// TIA Portal V16 export
// export: Created 2024-09-05T17:39:09.8002543Z, ExportSetting WithDefaults, DisplayName Totally Integrated Automation Portal, DisplayVersion V16 Update 6, DisplayName TIA Portal Version Control Interface, DisplayVersion V16 Update 2, DisplayName TIA Portal Openness, DisplayVersion V16 Update 6, DisplayName STEP 7 Professional, DisplayVersion V16 Update 6, DisplayName STEP 7 Safety, DisplayVersion V16, DisplayName WinCC Advanced, DisplayVersion V16 Update 6
FUNCTION_BLOCK "FittingCycle"   // FB35, LAD
{ S7_Optimized_Access := 'TRUE' }
VERSION : 0.1
// stored: AutoNumber true, IsIECCheckEnabled false, IsRetainMemResEnabled false, MemoryReserve 100, SetENOAutomatically false, UDAEnableTagReadback false
   VAR_INPUT
      parameters : "UDT_FittingParameters";
      basicPosition : Bool;
      MaxPosition : Real;
      endStopCylinderActive : Bool;
      shiftSupportToWork : Bool;
      rivetSensor : Bool;
      rivetStatusOtherCylinder : SInt;
   END_VAR
   VAR_IN_OUT
      HydraulicCylinder : "UDT_HydraulicCylinderData";
      dataFitting : "UDT_FittingStatus";
      dataDigiforce : "UDT_Digiforce";
      stopperForWedgeCylinder : "UDT_Cylinder";
      supportCylinder : "UDT_Cylinder";
      wedgeCylinder : "UDT_Cylinder";
      MeasuredData : "UDT_Results_Cupforming";
   END_VAR
   VAR
      cnt : Int;
      R_TRIG_Instance { S7_SetPoint := 'True'} : R_TRIG;
      H2Reached { S7_SetPoint := 'True'} : Bool;
      IEC_Timer_timeout { S7_SetPoint := 'True'} : TON_TIME;
      DigiforceStarted { S7_SetPoint := 'True'} : Bool;
      R_TRIG_Instance_1 { S7_SetPoint := 'True'} : R_TRIG;
      ton_WayWithTimeoutReached { S7_SetPoint := 'True'} : TON_TIME;
   END_VAR
   VAR_TEMP   // added for the SCL form of the ladder/FBD networks
      _w1 : Bool;
      _w2 : Bool;
   END_VAR
BEGIN

REGION Network 1: Check min max values
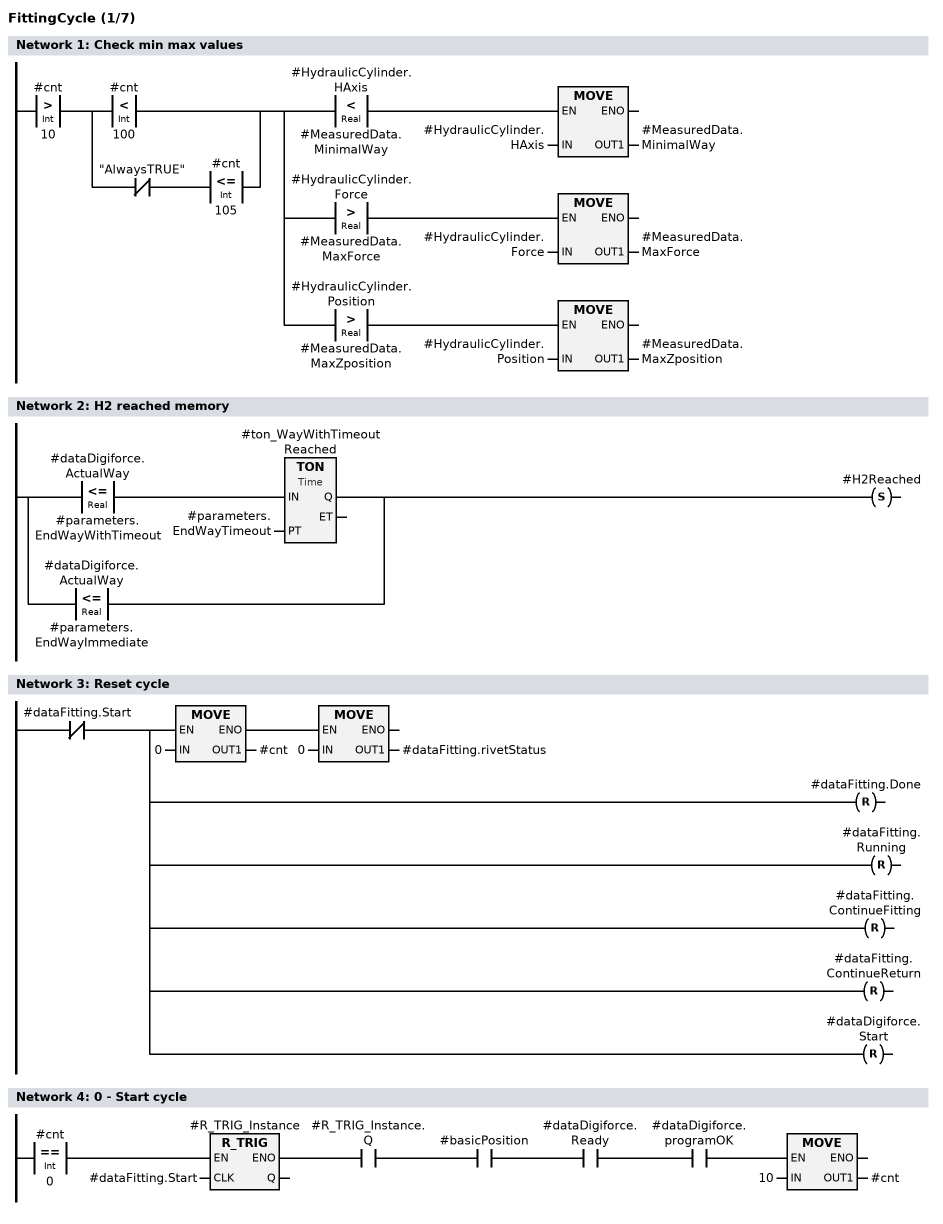
   RUNG wire#powerrail
      { S7_Templates := "SrcType := Int" } GT_Contact(in1 := #cnt, in2 := 10)
      wire#w1
      { S7_Templates := "SrcType := Int" } LT_Contact(in1 := #cnt, in2 := 100)
      wire#w2
      { S7_Templates := "SrcType := Real" } LT_Contact(in1 := #HydraulicCylinder.HAxis, in2 := #MeasuredData.MinimalWay)
      Move(in := #HydraulicCylinder.HAxis, out1 => #MeasuredData.MinimalWay)
   END_RUNG
   RUNG wire#w1
      I_Contact( "AlwaysTRUE" )
      { S7_Templates := "SrcType := Int" } LE_Contact(in1 := #cnt, in2 := 105)
   END_RUNG wire#w2
   RUNG wire#w2
      { S7_Templates := "SrcType := Real" } GT_Contact(in1 := #HydraulicCylinder.Force, in2 := #MeasuredData.MaxForce)
      Move(in := #HydraulicCylinder.Force, out1 => #MeasuredData.MaxForce)
   END_RUNG
   RUNG wire#w2
      { S7_Templates := "SrcType := Real" } GT_Contact(in1 := #HydraulicCylinder.Position, in2 := #MeasuredData.MaxZposition)
      Move(in := #HydraulicCylinder.Position, out1 => #MeasuredData.MaxZposition)
   END_RUNG
   // the same network as SCL:
   #_w1 := (#cnt > 10) AND ((#cnt < 100) OR (NOT "AlwaysTRUE" AND (#cnt <= 105)));
   IF #_w1 AND (#HydraulicCylinder.HAxis < #MeasuredData.MinimalWay) THEN
       #MeasuredData.MinimalWay := #HydraulicCylinder.HAxis;
   END_IF;
   IF #_w1 AND (#HydraulicCylinder.Force > #MeasuredData.MaxForce) THEN
       #MeasuredData.MaxForce := #HydraulicCylinder.Force;
   END_IF;
   IF #_w1 AND (#HydraulicCylinder.Position > #MeasuredData.MaxZposition) THEN
       #MeasuredData.MaxZposition := #HydraulicCylinder.Position;
   END_IF;
END_REGION

REGION Network 2: H2 reached memory
   RUNG wire#powerrail
      { S7_Templates := "SrcType := Real" } LE_Contact(in1 := #dataDigiforce.ActualWay, in2 := #parameters.EndWayWithTimeout)
      { S7_Templates := "time_type := Time" } #ton_WayWithTimeoutReached.TON(pt := #parameters.EndWayTimeout, et =>)
      wire#w1
      S_Coil( #H2Reached )
   END_RUNG
   RUNG wire#powerrail
      { S7_Templates := "SrcType := Real" } LE_Contact(in1 := #dataDigiforce.ActualWay, in2 := #parameters.EndWayImmediate)
   END_RUNG wire#w1
   // the same network as SCL:
   #ton_WayWithTimeoutReached(IN := #dataDigiforce.ActualWay <= #parameters.EndWayWithTimeout,   // TON
                           PT := #parameters.EndWayTimeout);
   IF #ton_WayWithTimeoutReached.Q OR (#dataDigiforce.ActualWay <= #parameters.EndWayImmediate) THEN
       #H2Reached := TRUE;
   END_IF;
END_REGION

REGION Network 3: Reset cycle
   RUNG wire#powerrail
      I_Contact( #dataFitting.Start )
      wire#w1
      Move(in := 0, out1 => #cnt)
      Move(in := 0, out1 => #dataFitting.rivetStatus)
   END_RUNG
   RUNG wire#w1
      R_Coil( #dataFitting.Done )
   END_RUNG
   RUNG wire#w1
      R_Coil( #dataFitting.Running )
   END_RUNG
   RUNG wire#w1
      R_Coil( #dataFitting.ContinueFitting )
   END_RUNG
   RUNG wire#w1
      R_Coil( #dataFitting.ContinueReturn )
   END_RUNG
   RUNG wire#w1
      R_Coil( #dataDigiforce.Start )
   END_RUNG
   // the same network as SCL:
   IF NOT #dataFitting.Start THEN
       #cnt := 0;
       #dataFitting.rivetStatus := 0;
       #dataFitting.Done := FALSE;
       #dataFitting.Running := FALSE;
       #dataFitting.ContinueFitting := FALSE;
       #dataFitting.ContinueReturn := FALSE;
       #dataDigiforce.Start := FALSE;
   END_IF;
END_REGION

REGION Network 4: 0 - Start cycle
   RUNG wire#powerrail
      { S7_Templates := "SrcType := Int" } EQ_Contact(in1 := #cnt, in2 := 0)
      #R_TRIG_Instance.R_TRIG(CLK := #dataFitting.Start, Q =>)
      Contact( #R_TRIG_Instance.Q )
      Contact( #basicPosition )
      Contact( #dataDigiforce.Ready )
      Contact( #dataDigiforce.programOK )
      Move(in := 10, out1 => #cnt)
   END_RUNG
   // the same network as SCL:
   #_w1 := #cnt = 0;
   #R_TRIG_Instance(EN := #_w1, CLK := #dataFitting.Start, ENO => #_w2);   // R_TRIG
   IF #_w2 AND #R_TRIG_Instance.Q AND #basicPosition AND #dataDigiforce.Ready AND #dataDigiforce.programOK THEN
       #cnt := 10;
   END_IF;
END_REGION

REGION Network 5: 10 - Start cycle
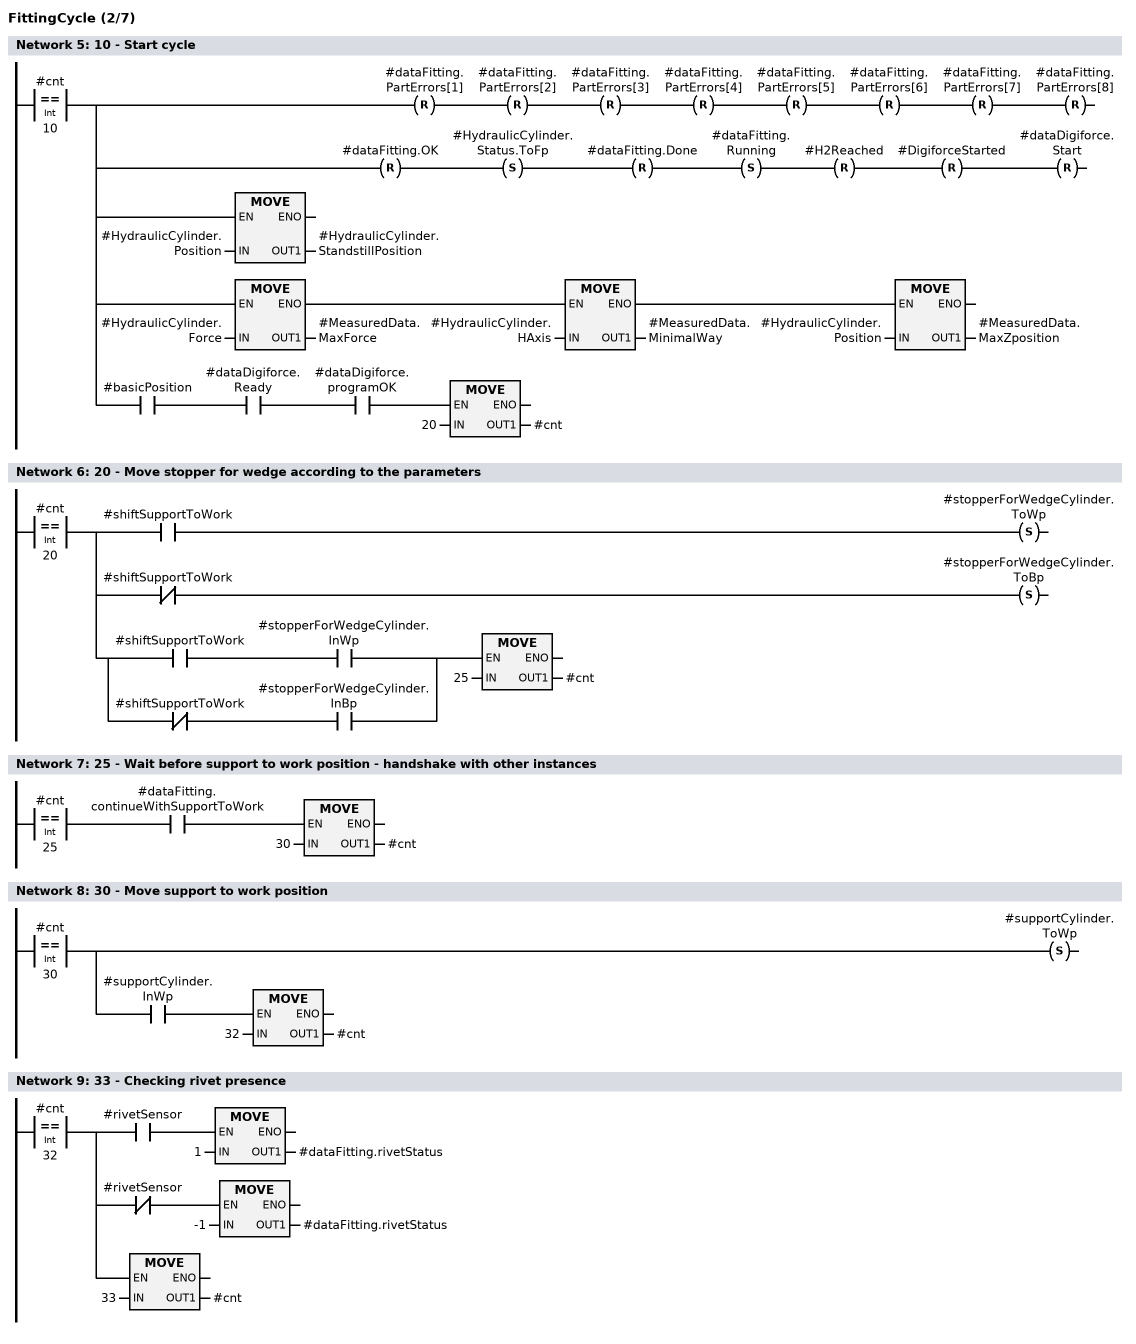
   RUNG wire#powerrail
      { S7_Templates := "SrcType := Int" } EQ_Contact(in1 := #cnt, in2 := 10)
      wire#w1
      R_Coil( #dataFitting.PartErrors[1] )
      R_Coil( #dataFitting.PartErrors[2] )
      R_Coil( #dataFitting.PartErrors[3] )
      R_Coil( #dataFitting.PartErrors[4] )
      R_Coil( #dataFitting.PartErrors[5] )
      R_Coil( #dataFitting.PartErrors[6] )
      R_Coil( #dataFitting.PartErrors[7] )
      R_Coil( #dataFitting.PartErrors[8] )
   END_RUNG
   RUNG wire#w1
      R_Coil( #dataFitting.OK )
      S_Coil( #HydraulicCylinder.Status.ToFp )
      R_Coil( #dataFitting.Done )
      S_Coil( #dataFitting.Running )
      R_Coil( #H2Reached )
      R_Coil( #DigiforceStarted )
      R_Coil( #dataDigiforce.Start )
   END_RUNG
   RUNG wire#w1
      Move(in := #HydraulicCylinder.Position, out1 => #HydraulicCylinder.StandstillPosition)
   END_RUNG
   RUNG wire#w1
      Move(in := #HydraulicCylinder.Force, out1 => #MeasuredData.MaxForce)
      Move(in := #HydraulicCylinder.HAxis, out1 => #MeasuredData.MinimalWay)
      Move(in := #HydraulicCylinder.Position, out1 => #MeasuredData.MaxZposition)
   END_RUNG
   RUNG wire#w1
      Contact( #basicPosition )
      Contact( #dataDigiforce.Ready )
      Contact( #dataDigiforce.programOK )
      Move(in := 20, out1 => #cnt)
   END_RUNG
   // the same network as SCL:
   #_w1 := #cnt = 10;
   IF #_w1 THEN
       #dataFitting.PartErrors[1] := FALSE;
       #dataFitting.PartErrors[2] := FALSE;
       #dataFitting.PartErrors[3] := FALSE;
       #dataFitting.PartErrors[4] := FALSE;
       #dataFitting.PartErrors[5] := FALSE;
       #dataFitting.PartErrors[6] := FALSE;
       #dataFitting.PartErrors[7] := FALSE;
       #dataFitting.PartErrors[8] := FALSE;
       #dataFitting.OK := FALSE;
       #HydraulicCylinder.Status.ToFp := TRUE;
       #dataFitting.Done := FALSE;
       #dataFitting.Running := TRUE;
       #H2Reached := FALSE;
       #DigiforceStarted := FALSE;
       #dataDigiforce.Start := FALSE;
       #HydraulicCylinder.StandstillPosition := #HydraulicCylinder.Position;
       #MeasuredData.MaxForce := #HydraulicCylinder.Force;
       #MeasuredData.MinimalWay := #HydraulicCylinder.HAxis;
       #MeasuredData.MaxZposition := #HydraulicCylinder.Position;
   END_IF;
   IF #_w1 AND #basicPosition AND #dataDigiforce.Ready AND #dataDigiforce.programOK THEN #cnt := 20; END_IF;
END_REGION

REGION Network 6: 20 - Move stopper for wedge according to the parameters
   RUNG wire#powerrail
      { S7_Templates := "SrcType := Int" } EQ_Contact(in1 := #cnt, in2 := 20)
      wire#w1
      Contact( #shiftSupportToWork )
      S_Coil( #stopperForWedgeCylinder.ToWp )
   END_RUNG
   RUNG wire#w1
      I_Contact( #shiftSupportToWork )
      S_Coil( #stopperForWedgeCylinder.ToBp )
   END_RUNG
   RUNG wire#w1
      Contact( #shiftSupportToWork )
      Contact( #stopperForWedgeCylinder.InWp )
      wire#w2
      Move(in := 25, out1 => #cnt)
   END_RUNG
   RUNG wire#w1
      I_Contact( #shiftSupportToWork )
      Contact( #stopperForWedgeCylinder.InBp )
   END_RUNG wire#w2
   // the same network as SCL:
   #_w1 := #cnt = 20;
   IF #_w1 AND #shiftSupportToWork THEN #stopperForWedgeCylinder.ToWp := TRUE; END_IF;
   IF #_w1 AND NOT #shiftSupportToWork THEN #stopperForWedgeCylinder.ToBp := TRUE; END_IF;
   IF #_w1 AND ((#shiftSupportToWork AND #stopperForWedgeCylinder.InWp) OR (NOT #shiftSupportToWork AND #stopperForWedgeCylinder.InBp)) THEN
       #cnt := 25;
   END_IF;
END_REGION

REGION Network 7: 25 - Wait before support to work position - handshake with other instances
   RUNG wire#powerrail
      { S7_Templates := "SrcType := Int" } EQ_Contact(in1 := #cnt, in2 := 25)
      Contact( #dataFitting.continueWithSupportToWork )
      Move(in := 30, out1 => #cnt)
   END_RUNG
   // the same network as SCL:
   IF (#cnt = 25) AND #dataFitting.continueWithSupportToWork THEN #cnt := 30; END_IF;
END_REGION

REGION Network 8: 30 - Move support to work position
   RUNG wire#powerrail
      { S7_Templates := "SrcType := Int" } EQ_Contact(in1 := #cnt, in2 := 30)
      wire#w1
      S_Coil( #supportCylinder.ToWp )
   END_RUNG
   RUNG wire#w1
      Contact( #supportCylinder.InWp )
      Move(in := 32, out1 => #cnt)
   END_RUNG
   // the same network as SCL:
   #_w1 := #cnt = 30;
   IF #_w1 THEN #supportCylinder.ToWp := TRUE; END_IF;
   IF #_w1 AND #supportCylinder.InWp THEN #cnt := 32; END_IF;
END_REGION

REGION Network 9: 33 - Checking rivet presence
   RUNG wire#powerrail
      { S7_Templates := "SrcType := Int" } EQ_Contact(in1 := #cnt, in2 := 32)
      wire#w1
      Contact( #rivetSensor )
      Move(in := 1, out1 => #dataFitting.rivetStatus)
   END_RUNG
   RUNG wire#w1
      I_Contact( #rivetSensor )
      Move(in := -1, out1 => #dataFitting.rivetStatus)
   END_RUNG
   RUNG wire#w1
      Move(in := 33, out1 => #cnt)
   END_RUNG
   // the same network as SCL:
   #_w1 := #cnt = 32;
   IF #_w1 AND #rivetSensor THEN #dataFitting.rivetStatus := 1; END_IF;
   IF #_w1 AND NOT #rivetSensor THEN #dataFitting.rivetStatus := -1; END_IF;
   IF #_w1 THEN #cnt := 33; END_IF;
END_REGION

REGION Network 10: 34 - Rivet presence result / handshake
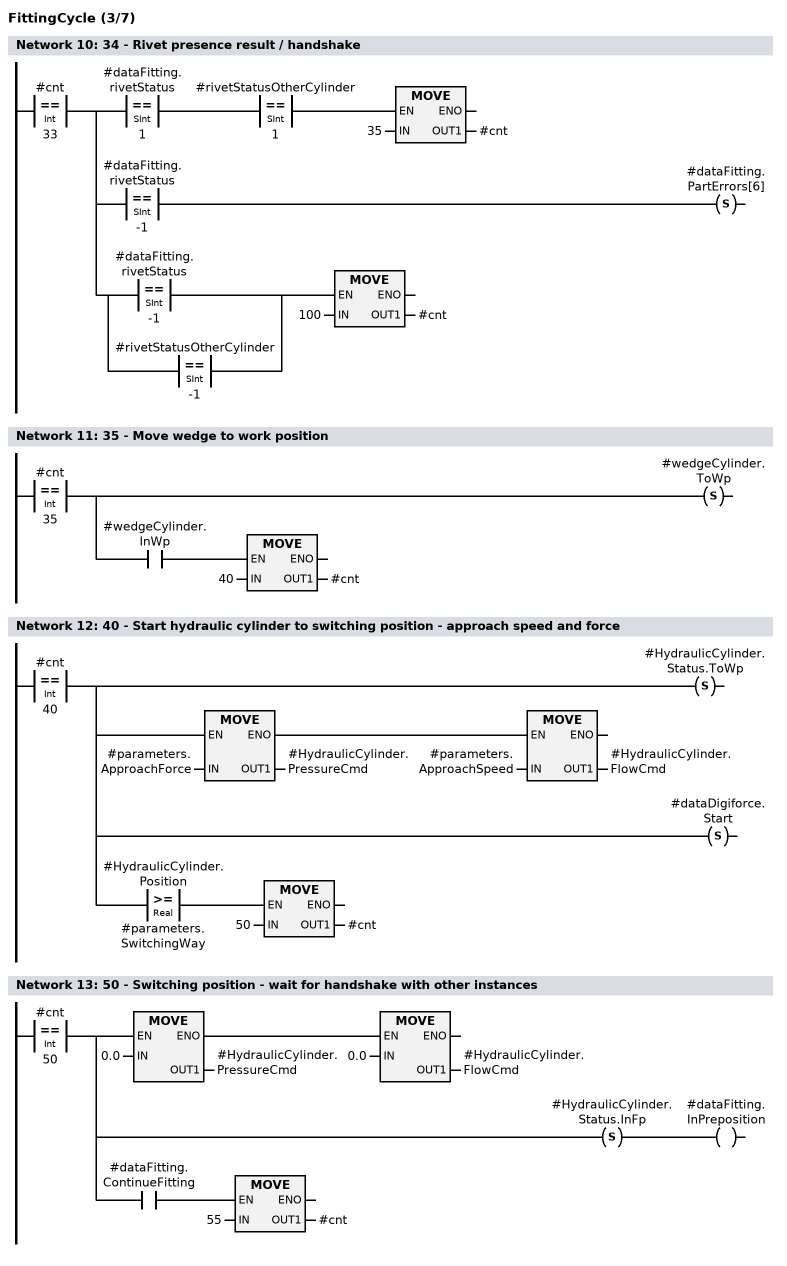
   RUNG wire#powerrail
      { S7_Templates := "SrcType := Int" } EQ_Contact(in1 := #cnt, in2 := 33)
      wire#w1
      { S7_Templates := "SrcType := SInt" } EQ_Contact(in1 := #dataFitting.rivetStatus, in2 := 1)
      { S7_Templates := "SrcType := SInt" } EQ_Contact(in1 := #rivetStatusOtherCylinder, in2 := 1)
      Move(in := 35, out1 => #cnt)
   END_RUNG
   RUNG wire#w1
      { S7_Templates := "SrcType := SInt" } EQ_Contact(in1 := #dataFitting.rivetStatus, in2 := -1)
      S_Coil( #dataFitting.PartErrors[6] )
   END_RUNG
   RUNG wire#w1
      { S7_Templates := "SrcType := SInt" } EQ_Contact(in1 := #dataFitting.rivetStatus, in2 := -1)
      wire#w2
      Move(in := 100, out1 => #cnt)
   END_RUNG
   RUNG wire#w1
      { S7_Templates := "SrcType := SInt" } EQ_Contact(in1 := #rivetStatusOtherCylinder, in2 := -1)
   END_RUNG wire#w2
   // the same network as SCL:
   #_w1 := #cnt = 33;
   IF #_w1 AND (#dataFitting.rivetStatus = 1) AND (#rivetStatusOtherCylinder = 1) THEN #cnt := 35; END_IF;
   IF #_w1 AND (#dataFitting.rivetStatus = (-1)) THEN #dataFitting.PartErrors[6] := TRUE; END_IF;
   IF #_w1 AND ((#dataFitting.rivetStatus = (-1)) OR (#rivetStatusOtherCylinder = (-1))) THEN
       #cnt := 100;
   END_IF;
END_REGION

REGION Network 11: 35 - Move wedge to work position
   RUNG wire#powerrail
      { S7_Templates := "SrcType := Int" } EQ_Contact(in1 := #cnt, in2 := 35)
      wire#w1
      S_Coil( #wedgeCylinder.ToWp )
   END_RUNG
   RUNG wire#w1
      Contact( #wedgeCylinder.InWp )
      Move(in := 40, out1 => #cnt)
   END_RUNG
   // the same network as SCL:
   #_w1 := #cnt = 35;
   IF #_w1 THEN #wedgeCylinder.ToWp := TRUE; END_IF;
   IF #_w1 AND #wedgeCylinder.InWp THEN #cnt := 40; END_IF;
END_REGION

REGION Network 12: 40 - Start hydraulic cylinder to switching position - approach speed and force
   RUNG wire#powerrail
      { S7_Templates := "SrcType := Int" } EQ_Contact(in1 := #cnt, in2 := 40)
      wire#w1
      S_Coil( #HydraulicCylinder.Status.ToWp )
   END_RUNG
   RUNG wire#w1
      Move(in := #parameters.ApproachForce, out1 => #HydraulicCylinder.PressureCmd)
      Move(in := #parameters.ApproachSpeed, out1 => #HydraulicCylinder.FlowCmd)
   END_RUNG
   RUNG wire#w1
      S_Coil( #dataDigiforce.Start )
   END_RUNG
   RUNG wire#w1
      { S7_Templates := "SrcType := Real" } GE_Contact(in1 := #HydraulicCylinder.Position, in2 := #parameters.SwitchingWay)
      Move(in := 50, out1 => #cnt)
   END_RUNG
   // the same network as SCL:
   #_w1 := #cnt = 40;
   IF #_w1 THEN
       #HydraulicCylinder.Status.ToWp := TRUE;
       #HydraulicCylinder.PressureCmd := #parameters.ApproachForce;
       #HydraulicCylinder.FlowCmd := #parameters.ApproachSpeed;
       #dataDigiforce.Start := TRUE;
   END_IF;
   IF #_w1 AND (#HydraulicCylinder.Position >= #parameters.SwitchingWay) THEN #cnt := 50; END_IF;
END_REGION

REGION Network 13: 50 - Switching position - wait for handshake with other instances
   RUNG wire#powerrail
      { S7_Templates := "SrcType := Int" } EQ_Contact(in1 := #cnt, in2 := 50)
      wire#w1
      Move(in := 0.0, out1 => #HydraulicCylinder.PressureCmd)
      Move(in := 0.0, out1 => #HydraulicCylinder.FlowCmd)
   END_RUNG
   RUNG wire#w1
      S_Coil( #HydraulicCylinder.Status.InFp )
      Coil( #dataFitting.InPreposition )
   END_RUNG
   RUNG wire#w1
      Contact( #dataFitting.ContinueFitting )
      Move(in := 55, out1 => #cnt)
   END_RUNG
   // the same network as SCL:
   #_w1 := #cnt = 50;
   IF #_w1 THEN
       #HydraulicCylinder.PressureCmd := 0.0;
       #HydraulicCylinder.FlowCmd := 0.0;
       #HydraulicCylinder.Status.InFp := TRUE;
   END_IF;
   #dataFitting.InPreposition := #_w1;
   IF #_w1 AND #dataFitting.ContinueFitting THEN #cnt := 55; END_IF;
END_REGION

REGION Network 14: 55 - Move sidemember to work position
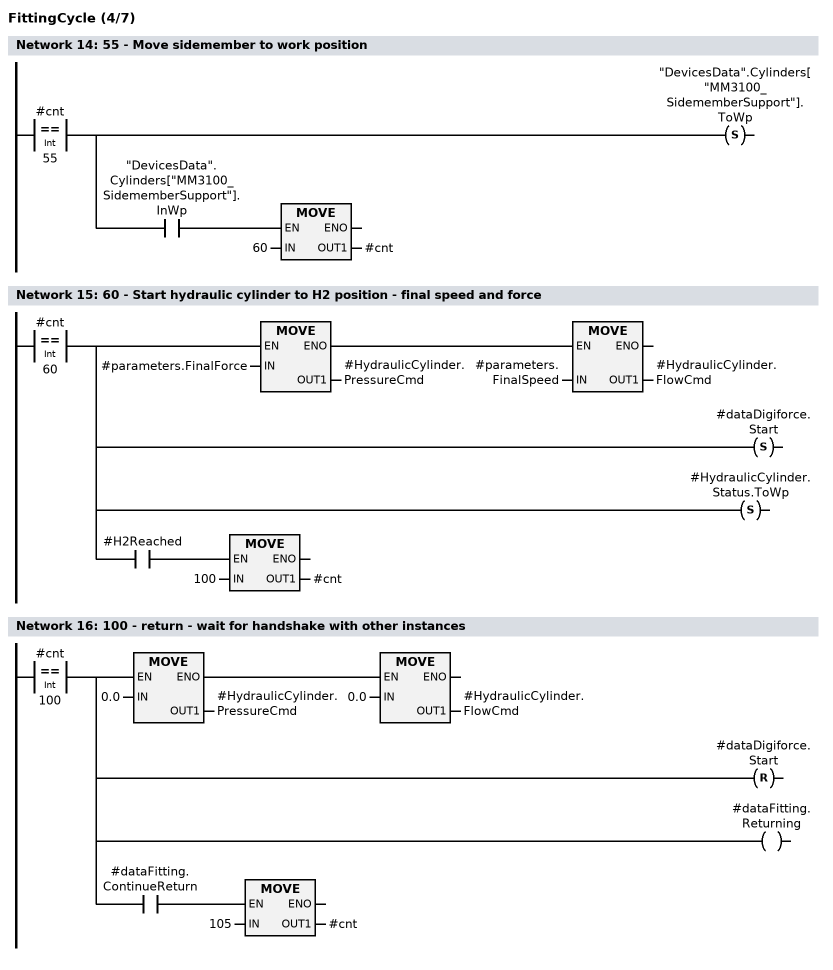
   RUNG wire#powerrail
      { S7_Templates := "SrcType := Int" } EQ_Contact(in1 := #cnt, in2 := 55)
      wire#w1
      S_Coil( "DevicesData".Cylinders["MM3100_SidememberSupport"].ToWp )
   END_RUNG
   RUNG wire#w1
      Contact( "DevicesData".Cylinders["MM3100_SidememberSupport"].InWp )
      Move(in := 60, out1 => #cnt)
   END_RUNG
   // the same network as SCL:
   #_w1 := #cnt = 55;
   IF #_w1 THEN "DevicesData".Cylinders["MM3100_SidememberSupport"].ToWp := TRUE; END_IF;
   IF #_w1 AND "DevicesData".Cylinders["MM3100_SidememberSupport"].InWp THEN #cnt := 60; END_IF;
END_REGION

REGION Network 15: 60 - Start hydraulic cylinder to H2 position - final speed and force
   RUNG wire#powerrail
      { S7_Templates := "SrcType := Int" } EQ_Contact(in1 := #cnt, in2 := 60)
      wire#w1
      Move(in := #parameters.FinalForce, out1 => #HydraulicCylinder.PressureCmd)
      Move(in := #parameters.FinalSpeed, out1 => #HydraulicCylinder.FlowCmd)
   END_RUNG
   RUNG wire#w1
      S_Coil( #dataDigiforce.Start )
   END_RUNG
   RUNG wire#w1
      S_Coil( #HydraulicCylinder.Status.ToWp )
   END_RUNG
   RUNG wire#w1
      Contact( #H2Reached )
      Move(in := 100, out1 => #cnt)
   END_RUNG
   // the same network as SCL:
   #_w1 := #cnt = 60;
   IF #_w1 THEN
       #HydraulicCylinder.PressureCmd := #parameters.FinalForce;
       #HydraulicCylinder.FlowCmd := #parameters.FinalSpeed;
       #dataDigiforce.Start := TRUE;
       #HydraulicCylinder.Status.ToWp := TRUE;
   END_IF;
   IF #_w1 AND #H2Reached THEN #cnt := 100; END_IF;
END_REGION

REGION Network 16: 100 - return - wait for handshake with other instances
   RUNG wire#powerrail
      { S7_Templates := "SrcType := Int" } EQ_Contact(in1 := #cnt, in2 := 100)
      wire#w1
      Move(in := 0.0, out1 => #HydraulicCylinder.PressureCmd)
      Move(in := 0.0, out1 => #HydraulicCylinder.FlowCmd)
   END_RUNG
   RUNG wire#w1
      R_Coil( #dataDigiforce.Start )
   END_RUNG
   RUNG wire#w1
      Coil( #dataFitting.Returning )
   END_RUNG
   RUNG wire#w1
      Contact( #dataFitting.ContinueReturn )
      Move(in := 105, out1 => #cnt)
   END_RUNG
   // the same network as SCL:
   #_w1 := #cnt = 100;
   IF #_w1 THEN
       #HydraulicCylinder.PressureCmd := 0.0;
       #HydraulicCylinder.FlowCmd := 0.0;
       #dataDigiforce.Start := FALSE;
   END_IF;
   #dataFitting.Returning := #_w1;
   IF #_w1 AND #dataFitting.ContinueReturn THEN #cnt := 105; END_IF;
END_REGION

REGION Network 17: 105 - Start returning
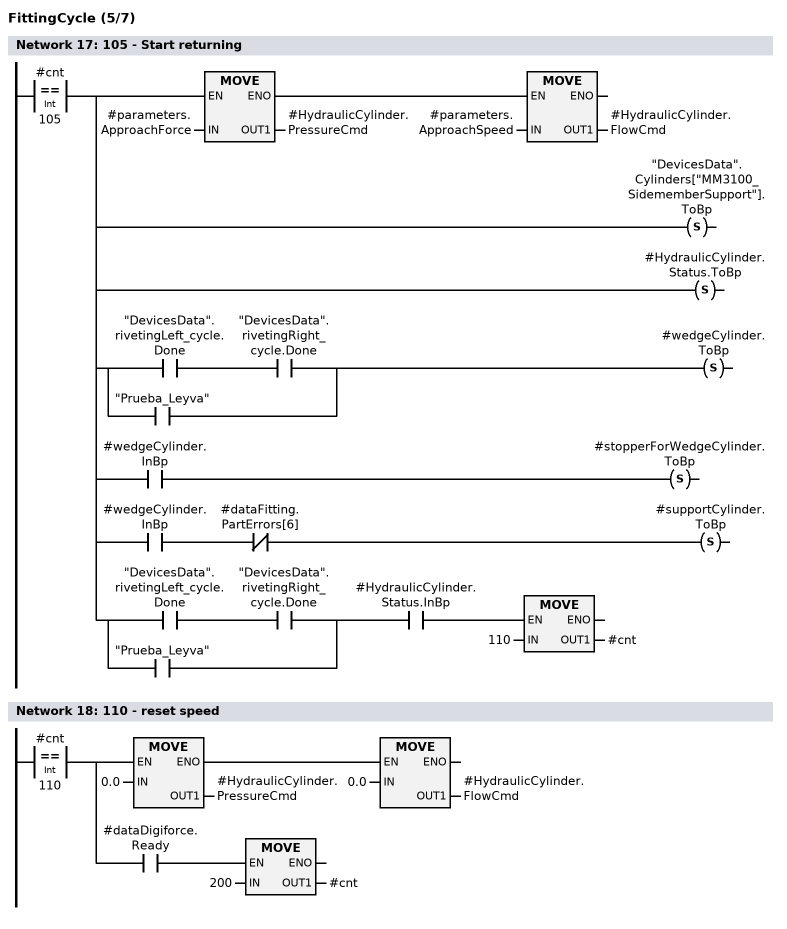
   RUNG wire#powerrail
      { S7_Templates := "SrcType := Int" } EQ_Contact(in1 := #cnt, in2 := 105)
      wire#w1
      Move(in := #parameters.ApproachForce, out1 => #HydraulicCylinder.PressureCmd)
      Move(in := #parameters.ApproachSpeed, out1 => #HydraulicCylinder.FlowCmd)
   END_RUNG
   RUNG wire#w1
      S_Coil( "DevicesData".Cylinders["MM3100_SidememberSupport"].ToBp )
   END_RUNG
   RUNG wire#w1
      S_Coil( #HydraulicCylinder.Status.ToBp )
   END_RUNG
   RUNG wire#w1
      Contact( "DevicesData".rivetingLeft_cycle.Done )
      Contact( "DevicesData".rivetingRight_cycle.Done )
      wire#w2
      S_Coil( #wedgeCylinder.ToBp )
   END_RUNG
   RUNG wire#w1
      Contact( "Prueba_Leyva" )
   END_RUNG wire#w2
   RUNG wire#w1
      Contact( #wedgeCylinder.InBp )
      S_Coil( #stopperForWedgeCylinder.ToBp )
   END_RUNG
   RUNG wire#w1
      Contact( #wedgeCylinder.InBp )
      I_Contact( #dataFitting.PartErrors[6] )
      S_Coil( #supportCylinder.ToBp )
   END_RUNG
   RUNG wire#w1
      Contact( "DevicesData".rivetingLeft_cycle.Done )
      Contact( "DevicesData".rivetingRight_cycle.Done )
      wire#w3
      Contact( #HydraulicCylinder.Status.InBp )
      Move(in := 110, out1 => #cnt)
   END_RUNG
   RUNG wire#w1
      Contact( "Prueba_Leyva" )
   END_RUNG wire#w3
   // the same network as SCL:
   #_w1 := #cnt = 105;
   IF #_w1 THEN
       #HydraulicCylinder.PressureCmd := #parameters.ApproachForce;
       #HydraulicCylinder.FlowCmd := #parameters.ApproachSpeed;
       "DevicesData".Cylinders["MM3100_SidememberSupport"].ToBp := TRUE;
       #HydraulicCylinder.Status.ToBp := TRUE;
   END_IF;
   IF #_w1 AND (("DevicesData".rivetingLeft_cycle.Done AND "DevicesData".rivetingRight_cycle.Done) OR "Prueba_Leyva") THEN
       #wedgeCylinder.ToBp := TRUE;
   END_IF;
   IF #_w1 AND #wedgeCylinder.InBp THEN #stopperForWedgeCylinder.ToBp := TRUE; END_IF;
   IF #_w1 AND #wedgeCylinder.InBp AND NOT #dataFitting.PartErrors[6] THEN
       #supportCylinder.ToBp := TRUE;
   END_IF;
   IF #_w1 AND (("DevicesData".rivetingLeft_cycle.Done AND "DevicesData".rivetingRight_cycle.Done) OR "Prueba_Leyva") AND #HydraulicCylinder.Status.InBp THEN
       #cnt := 110;
   END_IF;
END_REGION

REGION Network 18: 110 - reset speed
   RUNG wire#powerrail
      { S7_Templates := "SrcType := Int" } EQ_Contact(in1 := #cnt, in2 := 110)
      wire#w1
      Move(in := 0.0, out1 => #HydraulicCylinder.PressureCmd)
      Move(in := 0.0, out1 => #HydraulicCylinder.FlowCmd)
   END_RUNG
   RUNG wire#w1
      Contact( #dataDigiforce.Ready )
      Move(in := 200, out1 => #cnt)
   END_RUNG
   // the same network as SCL:
   #_w1 := #cnt = 110;
   IF #_w1 THEN
       #HydraulicCylinder.PressureCmd := 0.0;
       #HydraulicCylinder.FlowCmd := 0.0;
   END_IF;
   IF #_w1 AND #dataDigiforce.Ready THEN #cnt := 200; END_IF;
END_REGION

REGION Network 19: 200 - Move all cylinders to basic - evaluate result
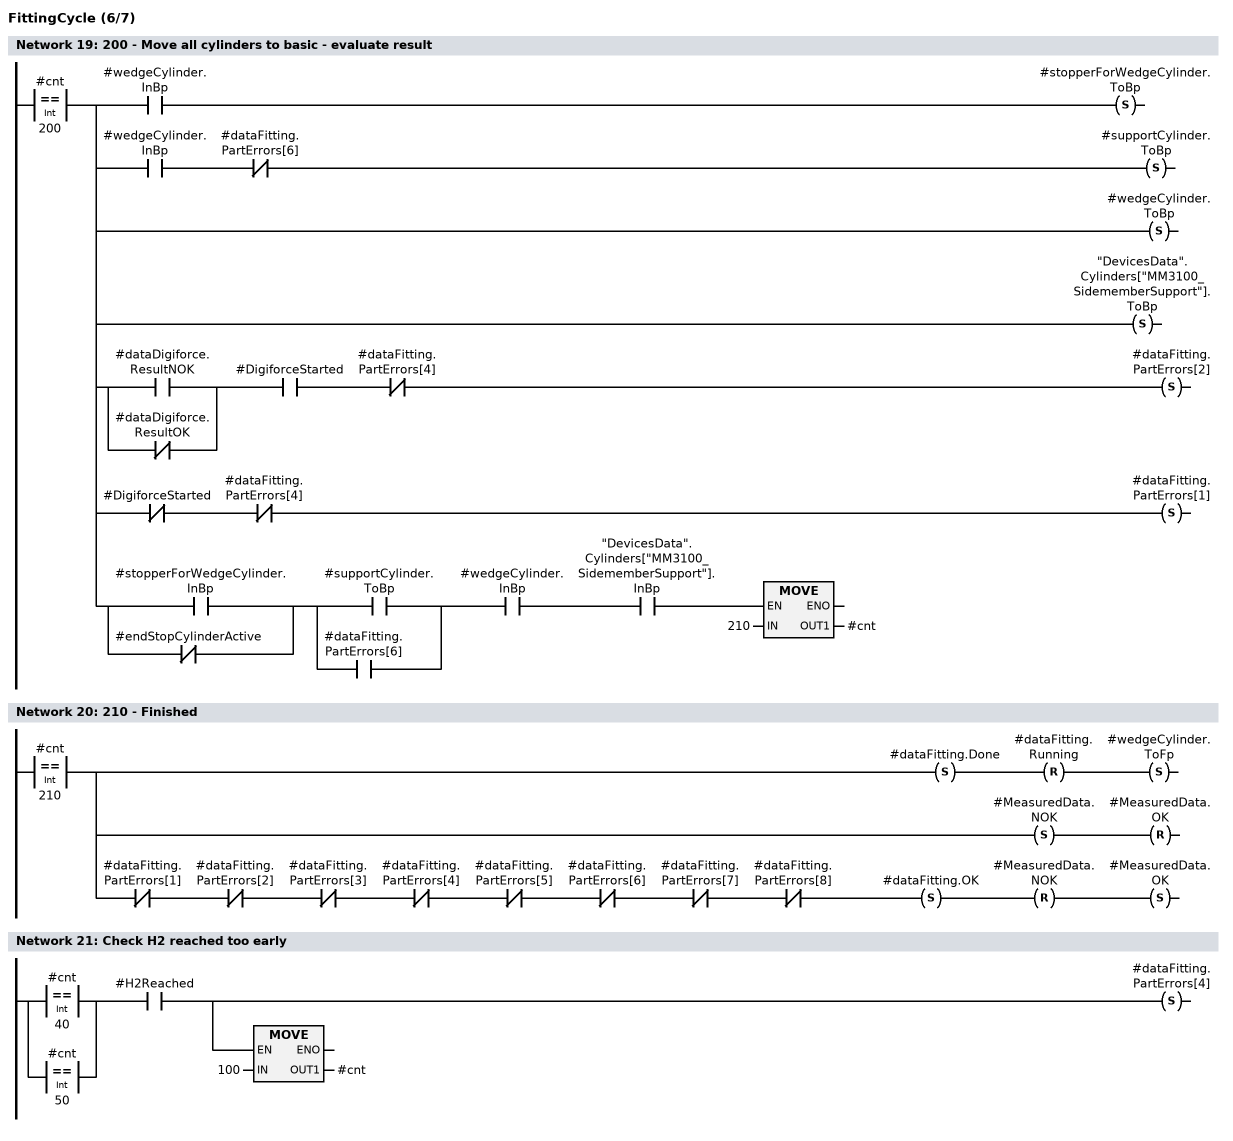
   RUNG wire#powerrail
      { S7_Templates := "SrcType := Int" } EQ_Contact(in1 := #cnt, in2 := 200)
      wire#w1
      Contact( #wedgeCylinder.InBp )
      S_Coil( #stopperForWedgeCylinder.ToBp )
   END_RUNG
   RUNG wire#w1
      Contact( #wedgeCylinder.InBp )
      I_Contact( #dataFitting.PartErrors[6] )
      S_Coil( #supportCylinder.ToBp )
   END_RUNG
   RUNG wire#w1
      S_Coil( #wedgeCylinder.ToBp )
   END_RUNG
   RUNG wire#w1
      S_Coil( "DevicesData".Cylinders["MM3100_SidememberSupport"].ToBp )
   END_RUNG
   RUNG wire#w1
      Contact( #dataDigiforce.ResultNOK )
      wire#w2
      Contact( #DigiforceStarted )
      I_Contact( #dataFitting.PartErrors[4] )
      S_Coil( #dataFitting.PartErrors[2] )
   END_RUNG
   RUNG wire#w1
      I_Contact( #dataDigiforce.ResultOK )
   END_RUNG wire#w2
   RUNG wire#w1
      I_Contact( #DigiforceStarted )
      I_Contact( #dataFitting.PartErrors[4] )
      S_Coil( #dataFitting.PartErrors[1] )
   END_RUNG
   RUNG wire#w1
      Contact( #stopperForWedgeCylinder.InBp )
      wire#w3
      Contact( #supportCylinder.ToBp )
      wire#w4
      Contact( #wedgeCylinder.InBp )
      Contact( "DevicesData".Cylinders["MM3100_SidememberSupport"].InBp )
      Move(in := 210, out1 => #cnt)
   END_RUNG
   RUNG wire#w1
      I_Contact( #endStopCylinderActive )
   END_RUNG wire#w3
   RUNG wire#w3
      Contact( #dataFitting.PartErrors[6] )
   END_RUNG wire#w4
   // the same network as SCL:
   #_w1 := #cnt = 200;
   IF #_w1 AND #wedgeCylinder.InBp THEN #stopperForWedgeCylinder.ToBp := TRUE; END_IF;
   IF #_w1 AND #wedgeCylinder.InBp AND NOT #dataFitting.PartErrors[6] THEN
       #supportCylinder.ToBp := TRUE;
   END_IF;
   IF #_w1 THEN
       #wedgeCylinder.ToBp := TRUE;
       "DevicesData".Cylinders["MM3100_SidememberSupport"].ToBp := TRUE;
   END_IF;
   IF #_w1 AND (#dataDigiforce.ResultNOK OR NOT #dataDigiforce.ResultOK) AND #DigiforceStarted AND NOT #dataFitting.PartErrors[4] THEN
       #dataFitting.PartErrors[2] := TRUE;
   END_IF;
   IF #_w1 AND NOT #DigiforceStarted AND NOT #dataFitting.PartErrors[4] THEN
       #dataFitting.PartErrors[1] := TRUE;
   END_IF;
   IF #_w1 AND (#stopperForWedgeCylinder.InBp OR NOT #endStopCylinderActive) AND (#supportCylinder.ToBp OR #dataFitting.PartErrors[6]) AND #wedgeCylinder.InBp AND "DevicesData".Cylinders["MM3100_SidememberSupport"].InBp THEN
       #cnt := 210;
   END_IF;
END_REGION

REGION Network 20: 210 - Finished
   RUNG wire#powerrail
      { S7_Templates := "SrcType := Int" } EQ_Contact(in1 := #cnt, in2 := 210)
      wire#w1
      S_Coil( #dataFitting.Done )
      R_Coil( #dataFitting.Running )
      S_Coil( #wedgeCylinder.ToFp )
   END_RUNG
   RUNG wire#w1
      S_Coil( #MeasuredData.NOK )
      R_Coil( #MeasuredData.OK )
   END_RUNG
   RUNG wire#w1
      I_Contact( #dataFitting.PartErrors[1] )
      I_Contact( #dataFitting.PartErrors[2] )
      I_Contact( #dataFitting.PartErrors[3] )
      I_Contact( #dataFitting.PartErrors[4] )
      I_Contact( #dataFitting.PartErrors[5] )
      I_Contact( #dataFitting.PartErrors[6] )
      I_Contact( #dataFitting.PartErrors[7] )
      I_Contact( #dataFitting.PartErrors[8] )
      S_Coil( #dataFitting.OK )
      R_Coil( #MeasuredData.NOK )
      S_Coil( #MeasuredData.OK )
   END_RUNG
   // the same network as SCL:
   #_w1 := #cnt = 210;
   IF #_w1 THEN
       #dataFitting.Done := TRUE;
       #dataFitting.Running := FALSE;
       #wedgeCylinder.ToFp := TRUE;
       #MeasuredData.NOK := TRUE;
       #MeasuredData.OK := FALSE;
   END_IF;
   IF #_w1 AND NOT #dataFitting.PartErrors[1] AND NOT #dataFitting.PartErrors[2] AND NOT #dataFitting.PartErrors[3] AND NOT #dataFitting.PartErrors[4] AND NOT #dataFitting.PartErrors[5] AND NOT #dataFitting.PartErrors[6] AND NOT #dataFitting.PartErrors[7] AND NOT #dataFitting.PartErrors[8] THEN
       #dataFitting.OK := TRUE;
       #MeasuredData.NOK := FALSE;
       #MeasuredData.OK := TRUE;
   END_IF;
END_REGION

REGION Network 21: Check H2 reached too early
   RUNG wire#powerrail
      { S7_Templates := "SrcType := Int" } EQ_Contact(in1 := #cnt, in2 := 40)
      wire#w1
      Contact( #H2Reached )
      wire#w2
      S_Coil( #dataFitting.PartErrors[4] )
   END_RUNG
   RUNG wire#powerrail
      { S7_Templates := "SrcType := Int" } EQ_Contact(in1 := #cnt, in2 := 50)
   END_RUNG wire#w1
   RUNG wire#w2
      Move(in := 100, out1 => #cnt)
   END_RUNG
   // the same network as SCL:
   IF ((#cnt = 40) OR (#cnt = 50)) AND #H2Reached THEN
       #dataFitting.PartErrors[4] := TRUE;
       #cnt := 100;
   END_IF;
END_REGION

REGION Network 22: Timeout
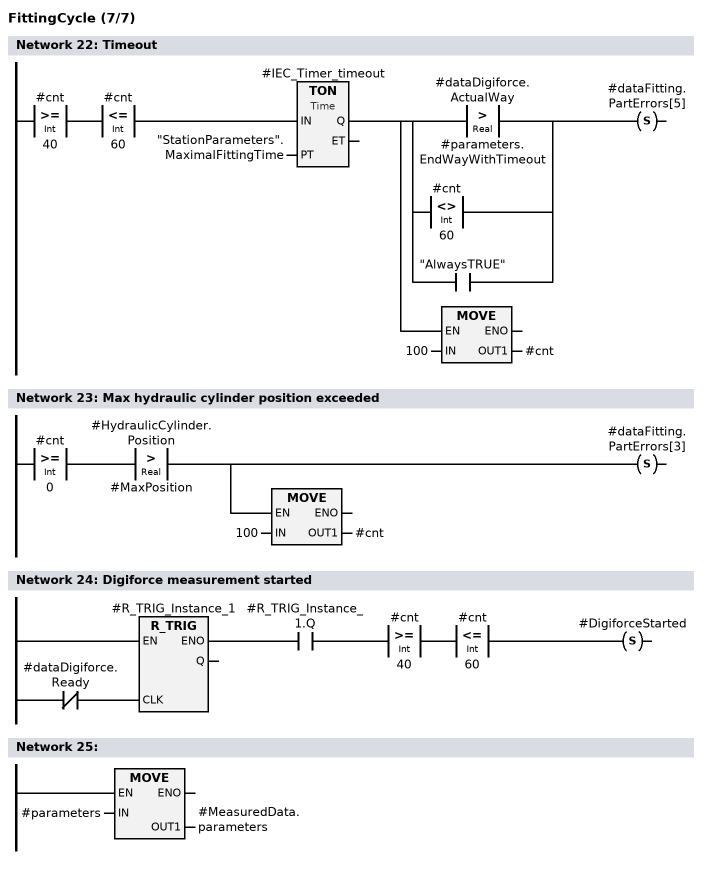
   RUNG wire#powerrail
      { S7_Templates := "SrcType := Int" } GE_Contact(in1 := #cnt, in2 := 40)
      { S7_Templates := "SrcType := Int" } LE_Contact(in1 := #cnt, in2 := 60)
      { S7_Templates := "time_type := Time" } #IEC_Timer_timeout.TON(pt := "StationParameters".MaximalFittingTime, et =>)
      wire#w1
      { S7_Templates := "SrcType := Real" } GT_Contact(in1 := #dataDigiforce.ActualWay, in2 := #parameters.EndWayWithTimeout)
      wire#w2
      S_Coil( #dataFitting.PartErrors[5] )
   END_RUNG
   RUNG wire#w1
      { S7_Templates := "SrcType := Int" } NE_Contact(in1 := #cnt, in2 := 60)
   END_RUNG wire#w2
   RUNG wire#w1
      Contact( "AlwaysTRUE" )
   END_RUNG wire#w2
   RUNG wire#w1
      Move(in := 100, out1 => #cnt)
   END_RUNG
   // the same network as SCL:
   #IEC_Timer_timeout(IN := (#cnt >= 40) AND (#cnt <= 60), PT := "StationParameters".MaximalFittingTime);   // TON
   IF #IEC_Timer_timeout.Q AND ((#dataDigiforce.ActualWay > #parameters.EndWayWithTimeout) OR (#cnt <> 60) OR "AlwaysTRUE") THEN
       #dataFitting.PartErrors[5] := TRUE;
   END_IF;
   IF #IEC_Timer_timeout.Q THEN #cnt := 100; END_IF;
END_REGION

REGION Network 23: Max hydraulic cylinder position exceeded
   RUNG wire#powerrail
      { S7_Templates := "SrcType := Int" } GE_Contact(in1 := #cnt, in2 := 0)
      { S7_Templates := "SrcType := Real" } GT_Contact(in1 := #HydraulicCylinder.Position, in2 := #MaxPosition)
      wire#w1
      S_Coil( #dataFitting.PartErrors[3] )
   END_RUNG
   RUNG wire#w1
      Move(in := 100, out1 => #cnt)
   END_RUNG
   // the same network as SCL:
   IF (#cnt >= 0) AND (#HydraulicCylinder.Position > #MaxPosition) THEN
       #dataFitting.PartErrors[3] := TRUE;
       #cnt := 100;
   END_IF;
END_REGION

REGION Network 24: Digiforce measurement started
   RUNG wire#powerrail
      #R_TRIG_Instance_1.R_TRIG(CLK := wire#w1, Q =>)
      Contact( #R_TRIG_Instance_1.Q )
      { S7_Templates := "SrcType := Int" } GE_Contact(in1 := #cnt, in2 := 40)
      { S7_Templates := "SrcType := Int" } LE_Contact(in1 := #cnt, in2 := 60)
      S_Coil( #DigiforceStarted )
   END_RUNG
   RUNG wire#powerrail
      I_Contact( #dataDigiforce.Ready )
   END_RUNG wire#w1
   // the same network as SCL:
   #R_TRIG_Instance_1(CLK := NOT #dataDigiforce.Ready, ENO => #_w1);   // R_TRIG
   IF #_w1 AND #R_TRIG_Instance_1.Q AND (#cnt >= 40) AND (#cnt <= 60) THEN #DigiforceStarted := TRUE; END_IF;
END_REGION

REGION Network 25
   RUNG wire#powerrail
      Move(in := #parameters, out1 => #MeasuredData.parameters)
   END_RUNG
   // the same network as SCL:
   #MeasuredData.parameters := #parameters;
END_REGION
END_FUNCTION_BLOCK
